{attribute 'linkalways'} 
{attribute 'no_explicit_call' := 'This FB is a CLASS and must be accessed using methods or properties'}
{attribute 'enable_dynamic_creation'}
FUNCTION_BLOCK Node_F_VN_InsertIntoContainer_INT EXTENDS VisionNode
VAR
    nElement : _INT(0);
    ipContainer : _ITcVnContainer;
    nIndex : _ULINT(0);
    hrPrev : _HRESULT(S_OK);
    hresult : _HRESULT(S_OK);
END_VAR

METHOD PUBLIC  Clone : I_Node
VAR
	pNode : POINTER TO Node_F_VN_InsertIntoContainer_INT;
END_VAR
pNode := __NEW(Node_F_VN_InsertIntoContainer_INT);
Clone := pNode^;
END_METHOD

METHOD FB_init : BOOL
VAR_INPUT
	bInitRetains : BOOL; // if TRUE, the retain variables are initialized (warm start / cold start)
	bInCopyCode : BOOL;  // if TRUE, the instance afterwards gets moved into the copy code (online change)
END_VAR
AddInput('nElement', nElement);
AddInput('ipContainer', ipContainer);
AddInput('nIndex', nIndex);
AddInput('hrPrev', hrPrev);
AddOutput('ipContainer', ipContainer);
AddOutput('hresult',hresult);
END_METHOD

METHOD PROTECTED OnExecute : HRESULT
hresult.Value := F_VN_InsertIntoContainer_INT(
    nElement := nElement.Value,
    ipContainer := ipContainer.Value,
    nIndex := nIndex.Value,
    hrPrev:= hrPrev.Value);
END_METHOD

METHOD PUBLIC PreExecutionCheck
VAR_INPUT
	Check : I_PreExecutionChecks;
END_VAR
Check.IsTrue(ipContainer.IsValid, 'ipContainer must be a valid container');
END_METHOD

END_FUNCTION_BLOCK

(* stored: Version 1.1.0.1, ProductVersion 3.1.4024.13
   POU Node_F_VN_InsertIntoContainer_INT: Id {935b7b2b-6f5d-46f0-b97f-3a2ece65b2ca}, SpecialFunc None
   Folder Constructor: Id {19173e89-fefd-42f4-92c2-9883cf0f0cd4}
   Method Clone: Id {a8c2a035-0b61-4cb3-a99a-4eeba0f27cfb}
   Method FB_init: Id {06f87a77-82b4-4c2a-ab0d-c006c482478a}
   Method OnExecute: Id {1e5c8891-c73d-4523-9ac8-ef3b02a83f54}
   Method PreExecutionCheck: Id {b9a9bce4-75c4-4975-a680-703312f6a230} *)
